Staubli VAL3: buildList.pgx

program buildList()
  local num l_nSize
  local InstrItem l_iEvent
  local num i
  local string l_sEmpty
  local num l_nResult
  local num l_nSizeItem
  local num j
  local TrajectoryItem l_tTraj
  local string l_sPath
  local num k
  local progItem l_pProg
  local string l_sData
  local string l_sType
begin
  // INIT the list
  l_sEmpty=""
  call use:stringCopy(l_sEmpty,sList)
  // add the items
  call prog:getSizeItem(l_nSize)
  for i=0 to (l_nSize-1)
    call prog:getItem(l_iEvent,i)
    if l_iEvent.sType!=""
      l_sData=l_iEvent.sData
      l_sType=l_iEvent.sType
      call saveInputOutput:replaceIO(l_sData,l_sType,l_sData)
      call listAdd(toString("2",i+1)+" "+l_sType+" "+l_sData)
      if find(l_iEvent.sType,"#")!=-1
        l_iEvent.sType=right(l_iEvent.sType,len(l_iEvent.sType)-1)
      endIf
      // show the name of IN OUT NUM
      if saveData:bShowItem and find(l_iEvent.sData,"@")==-1
        // get inside the trajectory field
        call saveData:getPathInstr(l_iEvent.sType,l_sPath)
        // TRAJECTORY
        if TrajItem:libLoad(l_sPath)==0
          delay(0)
          // scan for the action
          call TrajItem:load(l_iEvent.sData,l_nResult)
          if l_nResult==0
            call TrajItem:getSizeItem(false,l_nSizeItem)
            // patch for the PALLET
            if find(TrajItem:libPath(),"PALLET")!=-1
              l_nSizeItem=1
            endIf
            // scan for the TCP
            for j=0 to l_nSizeItem-1
              call TrajItem:getTrajItem(l_tTraj,j)
              // scan for the TCP
              if l_tTraj.nTcpAction==1
                call listAdd("  -TCP ON ")
              elseIf l_tTraj.nTcpAction==2
                call listAdd("  -TCP OFF ")
              endIf
              for k=0 to size(l_tTraj.iInstr)-1
                if l_tTraj.iInstr[k].sType!=""
                  l_sData=l_tTraj.iInstr[k].sData
                  l_sType=l_tTraj.iInstr[k].sType
                  call saveInputOutput:replaceIO(l_sData,l_sType,l_sData)
                  call listAdd("   -"+l_sType+" "+l_sData)
                endIf
              endFor
            endFor
          endIf
        elseIf l_iEvent.sType=="SUB"
          // SUB
          call sub:load(l_iEvent.sData,l_nResult)
          if l_nResult==0
            call sub:getProgItem(l_pProg,l_iEvent.sData)
            l_nSizeItem=size(l_pProg.iEvent)
            for j=0 to l_nSizeItem-1
              if l_pProg.iEvent[j].sType!=""
                l_sData=l_pProg.iEvent[j].sData
                l_sType=l_pProg.iEvent[j].sType
                call saveInputOutput:replaceIO(l_sData,l_sType,l_sData)
                call listAdd("  -"+l_sType+" "+l_sData)
              endIf
            endFor
          endIf
        endIf
      endIf
    else
      // delete empty space
      call prog:deleteItem(i,l_nResult)
      // recovery
      call prog:getSizeItem(l_nSize)
      i=i-1
    endIf
  endFor
  //
  use:bUseRefresh=true
end
